PROGRAM Safety
VAR
END_VAR

// Safety for Rotation:
IF Automatic.RotationPositionCurrent >= 570 AND NOT IO.ButtonLowerLeft THEN
	//IO.MotorRotation := 0;
	//Automatic.MotorR.CurrentlyMoving := FALSE;
END_IF
IF IO.EndRotationSensor THEN
	Automatic.RotationPositionCurrent := 0;
	Automatic.MotorR.CurrentlyMoving := FALSE;
END_IF

// Safety for Lifting:
IF Automatic.LiftingPositionCurrent >= 355 AND NOT IO.ButtonLowerLeft THEN
	//IO.MotorLifting := 0;
	// Automatic.MotorL.CurrentlyMoving := FALSE;
END_IF
IF IO.EndLiftingSensor THEN
	Automatic.LiftingPositionCurrent := 0;
	Automatic.MotorL.CurrentlyMoving := FALSE;
END_IF

// Safety for Extension:
IF Automatic.ExtensionPositionCurrent >= 445 AND NOT IO.ButtonLowerLeft THEN
	//IO.MotorExtension := 0;
	//Automatic.MotorE.CurrentlyMoving := FALSE;
END_IF
IF IO.EndExtensionSensor THEN
	Automatic.ExtensionPositionCurrent := 0;
	Automatic.MotorE.CurrentlyMoving := FALSE;
END_IF

// Safety for Grip:
IF Automatic.GripPositionCurrent >= 80 AND NOT IO.ButtonLowerLeft THEN
	//IO.MotorGrip := 0;
	// Automatic.MotorG.CurrentlyMoving := FALSE;
END_IF
IF IO.EndGripSensor THEN
	Automatic.GripPositionCurrent := 0;
	Automatic.MotorG.CurrentlyMoving := FALSE;
END_IF

END_PROGRAM

(* stored: Version 1.1.0.1, ProductVersion 3.1.4024.13
   POU Safety: Id {8bf2167f-22d8-4543-8367-d7ef70615958}, SpecialFunc None *)
